// TIA Portal V18 export
DATA_BLOCK "FB23-regenarationpgmFB_DB"   // DB178
VERSION : 0.1
// stored: AutoNumber true, DBAccessibleFromOPCUA true, InstanceOfName FB23-regenarationpgmFB, InstanceOfType FB
"FB23-regenarationpgmFB"
   // VAR_INPUT
   //    Dispensing_time : DInt;
   //    "Set Qty in ml" : Real;
   //    "Pump ON A delay" : DInt;
   //    "Pump ON B delay" : DInt;
   //    "Mixer Off delay" : DInt;
   // END_VAR
   // VAR_OUTPUT
   //    "Run time" : Int;
   // END_VAR
   // VAR_IN_OUT
   //    ON_Pump_A : Bool;
   //    ON_pump_B : Bool;
   //    ON_Mixer : Bool;
   //    "Start Metering" : Bool;
   //    "Stop metering" : Bool;
   //    "Process running" : Bool;
   //    "process completed" : Bool;
   // END_VAR
   // VAR
   //    "Total Volume dispensed" : Real;
   //    "metering started" : Bool;
   //    "metering time in msec" : DInt;
   //    "dispense time elapsed" : Bool;
   // END_VAR
BEGIN
END_DATA_BLOCK
